FUNCTION INTERNAL F_ReadRepeatedField : HRESULT
VAR_IN_OUT      
    stCtx : ST_ParseContext;
END_VAR
VAR_INPUT CONSTANT
    anyArray        : T_Any;
    anyFirstElem    : T_Any;
    ipFieldCodec    : I_FieldCodec; 
END_VAR

VAR_IN_OUT   
    nFieldIndex : UDINT; 
END_VAR
VAR
    nTag        : UDINT;
    hr          : HRESULT;
    nLength     : UDINT;
    nCurrentLimit : UDINT;
    nArrayLength: UDINT;
    nByteLength : UDINT;
    nTypeSize   : UDINT;
    bTagConsumed: BOOL;
    nBufferEnd  : UDINT;  
    anyValue    : T_ANY;
END_VAR

IF ipFieldCodec = 0 THEN
    F_ReadRepeatedField := F_ParseError(stCtx,  E_ParserErrorCode.InternalError);
    RETURN;
END_IF

IF anyArray.TypeClass <> __SYSTEM.TYPE_CLASS.TYPE_ARRAY THEN
    F_ReadRepeatedField := F_ParseError(stCtx, E_ParserErrorCode.InvalidDataType);
    RETURN;
END_IF

nTypeSize := TO_UDINT(anyFirstElem.diSize);

IF nTypeSize = 0 THEN
    F_ReadRepeatedField :=  F_ParseError(stCtx, E_ParserErrorCode.InvalidDataType);
    RETURN;
END_IF

nByteLength := TO_UDINT(anyArray.diSize);
nArrayLength := nByteLength / nTypeSize;

nTag := stCtx.stState.nLastTag;

IF  nFieldIndex < 0 OR nFieldIndex >= nArrayLength THEN
    F_ReadRepeatedField :=  F_ParseError(stCtx, E_ParserErrorCode.NotEnoughMem);
    RETURN;
END_IF

IF ipFieldCodec.IsPackedRepeatedField(nTag) THEN
    
    hr := F_ParseLength(stCtx, nLength=> nLength);
    IF FAILED(hr) OR nLength <= 0 THEN
        // Empty packed field, valid - ignore.
        F_ReadRepeatedField := hr;
        RETURN;
    END_IF 
    
    F_SbhPushLimit(stCtx.stState, nLength, nCurrentLimit=> nCurrentLimit);
    nBufferEnd := stCtx.stState.nBufferPos + nLength;
    WHILE NOT F_SbhIsReachedLimit(stCtx.stState) DO
        hr := ipFieldCodec.ValueReader(stCtx, anyOut=> anyValue);
        IF FAILED(hr) THEN
            F_ReadRepeatedField := hr;
            RETURN;
        END_IF
        
        MEMCPY(destAddr:= anyArray.pValue + (nFieldIndex * nTypeSize), srcAddr:= anyValue.pValue, MIN(TO_UDINT(anyValue.diSize), nTypeSize));
        nFieldIndex := nFieldIndex + 1;
    END_WHILE

    F_SbhPopLimit(stCtx.stState, nCurrentLimit);
ELSE
    // Not packed or possibly not packable...
    REPEAT
        hr := ipFieldCodec.ValueReader(stCtx, anyOut=> anyValue);
        IF FAILED(hr) THEN
            F_ReadRepeatedField := hr;
            RETURN;
        END_IF
        
        MEMCPY(destAddr:= anyArray.pValue + (nFieldIndex * nTypeSize), srcAddr:= anyValue.pValue, MIN(TO_UDINT(anyValue.diSize), nTypeSize));
        nFieldIndex := nFieldIndex + 1;
        
        hr := F_MaybeConsumeTag(stCtx, nTag, bConsumed=> bTagConsumed);
        IF FAILED(hr) THEN
            F_ReadRepeatedField := hr;
            RETURN;
        END_IF
    UNTIL
        NOT bTagConsumed
    END_REPEAT
END_IF

END_FUNCTION

(* stored: Version 1.1.0.1
   POU F_ReadRepeatedField: Id {3275937c-bc24-42b8-bf5d-84307b144b13}, SpecialFunc None *)
